Universal Robots PolyScope program: socket.urp

ProgramRoot directory=/home/ur/ursim-3.1/programs/36-socket; kinematics=(a=[0, -0.425, -0.39225, 0, 0, 0], d=[0.08916, 0, 0, 0.10915, 0.09465, 0.0823], alpha=[1.5708, 0, 0, 1.5708, -1.5708, 0], deltaTheta=[0, 0, 0, 0, 0, 0], status=notInitialized); lastSavedInVersion=(project__name=Polyscope, major__version=3, minor__version=1, svn__revision=17195, build__date=Mar 11 2015, 13:02:28); name=socket; programVersion=(project__name=Polyscope, major__version=3, minor__version=1, svn__revision=17195, build__date=Mar 11 2015, 13:02:28); robotEnvironmentFileName=default; serialNumberRobot=2014350001
  BeforeStart description=COMMAND_SEQUENCE_BEFORE_PROGRAM_START; name=BeforeStart
    Assignment expr=socket_open("192.168.1.7",30000); operatorValueType=INTEGER; valueSource=EXPRESSION
    While count=0; expr=ExpressionVariableNode≟ False; type=LOOP_EXPR
      Assignment expr=socket_open("192.168.1.7",30000); operatorValueType=INTEGER; valueSource=EXPRESSION
      Script type=0; expressionBranchNode=sync()
  MainProgram cartesianAcceleration=1.2; cartesianSpeed=0.25; jointAcceleration=1.3962634015954636; jointSpeed=1.0471975511965976; sharedProcessMoveBlendRadius=0.025; motionType=JOINT_SPACE
    Assignment expr=socket_read_ascii_float(6); operatorValueType=INTEGER; valueSource=EXPRESSION
    If expr=ExpressionVariableNode[0]≟6; type=IF_NODE
      Script type=0; expressionBranchNode=socket_send_line("received")
